(* Logix 5000 project; controller IF2_DEMO Emulate 5570 rev 20.12; software revision 20.04; part 4 of 8 *)
(* tags used below, declared in another part *)
   Alarm_Labeler1_Blocked : ALARM_DIGITAL;
   Alarm_Labeler1_Breakdown : ALARM_DIGITAL;
   Alarm_Labeler1_Starved : ALARM_DIGITAL;
   Alarm_Labeler1_Stopped : ALARM_DIGITAL;
   Blocked_Condition : BOOL;
   Breakdown_Labeler_Simulation : TIMER;
   Breakdown_Labeler_Simulator_Down_Switch : BOOL;
   Breakdown_Occurance_Time : DINT;
   Breakdown_Variation_Stepper : DINT;
   Expected_Full_Production_Rate : DINT;
   Labeler : FTVPDemoWorkCell;
   Labeler_Bottler_Per_Min : DINT;
   Labeler_Start : BOOL;
   Labeler_State : DINT;
   Labeler_Status : DINT;
   Labeler_Stop : BOOL;
   OEE_Availability : REAL;
   OEE_Overall : REAL;
   OEE_Performance : REAL;
   OEE_Quality : REAL;
   Starve_Block_Labeler_ONS : BOOL;
   Starved_Condition : BOOL;
   TempReadTrigger : TIMER;
   TempTimer : TIMER;
   TempTimer2 : TIMER;
   AlarmLabelJam : BOOL;
   ChangeOver_In_Progress : BOOL;
   Current_Order : STRING;
   CurrentCustomerName : STRING;
   CurrentPartName : STRING;
   DispenserLine : LineData;
   Filler_Bottles_Per_Minute : ALIAS FOR ProdCounts.Total;
   Filler_Stopped : BOOL;
   Labeler_Stopped : BOOL;
   OEE_Scrap_Labeler : DINT;
   OrderQty : DINT[4];
   Packaging_Stopped : BOOL;
   PartCountRollOver : DINT;
   Performance_Control : DINT;
   Previous_Order : STRING;
   PreviousCustomerName : STRING;
   PreviousPartName : STRING;
   ProdCounts : Counts;
   Product_Change : DINT;
   Production_Start_Labeler : BOOL;
   RefillLine : LineData;
   Starve_Block_Filler_Start_Toggle : BOOL;
   Starve_Block_Labeler_Start_Toggle : BOOL;
   Starve_Block_Packaging_Start_Toggle : BOOL;
   Timer1000ms : TIMER;
   Timer250ms : TIMER;
   WallClock : DINT[7];
   WC : WC[10];
(* LabelerD, continued *)

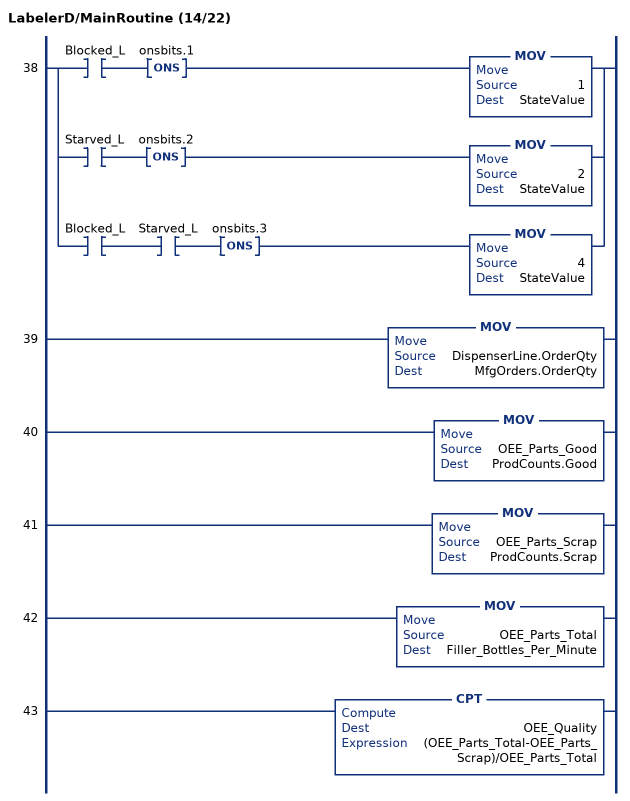
   38: [XIC(Blocked_L) ONS(onsbits.1) MOV(1,StateValue) ,XIC(Starved_L) ONS(onsbits.2) MOV(2,StateValue) ,XIC(Blocked_L) XIC(Starved_L) ONS(onsbits.3) MOV(4,StateValue) ];
   39: MOV(DispenserLine.OrderQty,MfgOrders.OrderQty);
   40: MOV(OEE_Parts_Good,ProdCounts.Good);
   41: MOV(OEE_Parts_Scrap,ProdCounts.Scrap);
   42: MOV(OEE_Parts_Total,Filler_Bottles_Per_Minute);
   43: CPT(OEE_Quality,(OEE_Parts_Total-OEE_Parts_Scrap)/OEE_Parts_Total);
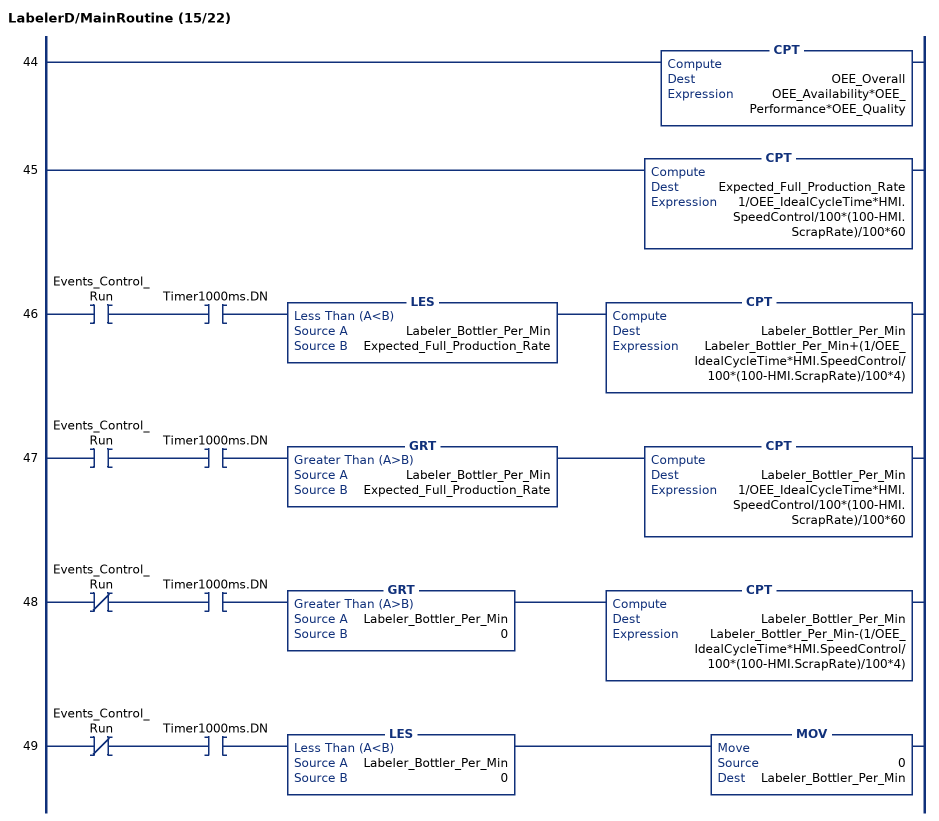
   44: CPT(OEE_Overall,OEE_Availability*OEE_Performance*OEE_Quality);
   45: CPT(Expected_Full_Production_Rate,1/OEE_IdealCycleTime*HMI.SpeedControl/100*(100-HMI.ScrapRate)/100*60);
   46: XIC(Events_Control_Run)XIC(Timer1000ms.DN)LES(Labeler_Bottler_Per_Min,Expected_Full_Production_Rate)CPT(Labeler_Bottler_Per_Min,Labeler_Bottler_Per_Min+(1/OEE_IdealCycleTime*HMI.SpeedControl/100*(100-HMI.ScrapRate)/100*4));
   47: XIC(Events_Control_Run)XIC(Timer1000ms.DN)GRT(Labeler_Bottler_Per_Min,Expected_Full_Production_Rate)CPT(Labeler_Bottler_Per_Min,1/OEE_IdealCycleTime*HMI.SpeedControl/100*(100-HMI.ScrapRate)/100*60);
   48: XIO(Events_Control_Run)XIC(Timer1000ms.DN)GRT(Labeler_Bottler_Per_Min,0)CPT(Labeler_Bottler_Per_Min,Labeler_Bottler_Per_Min-(1/OEE_IdealCycleTime*HMI.SpeedControl/100*(100-HMI.ScrapRate)/100*4));
   49: XIO(Events_Control_Run)XIC(Timer1000ms.DN)LES(Labeler_Bottler_Per_Min,0)MOV(0,Labeler_Bottler_Per_Min);
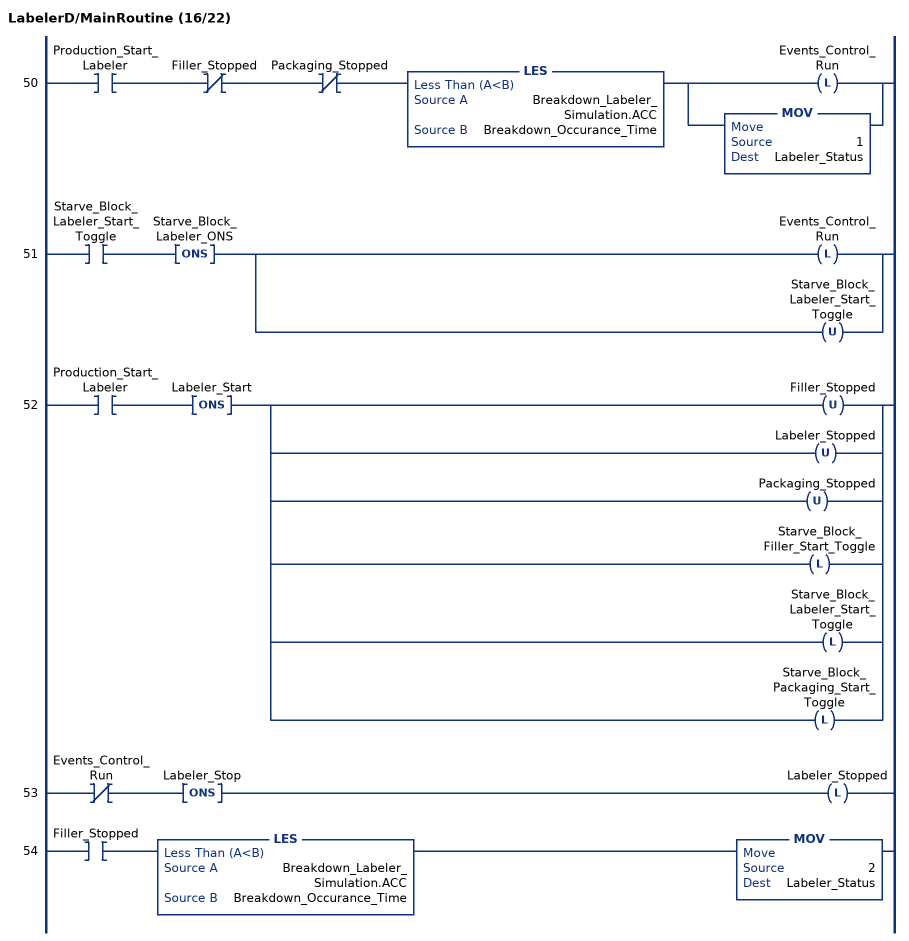
   50: XIC(Production_Start_Labeler)XIO(Filler_Stopped)XIO(Packaging_Stopped)LES(Breakdown_Labeler_Simulation.ACC,Breakdown_Occurance_Time)[OTL(Events_Control_Run) ,MOV(1,Labeler_Status) ];
   51: XIC(Starve_Block_Labeler_Start_Toggle)ONS(Starve_Block_Labeler_ONS)[OTL(Events_Control_Run) ,OTU(Starve_Block_Labeler_Start_Toggle) ];
   52: XIC(Production_Start_Labeler)ONS(Labeler_Start)[OTU(Filler_Stopped) ,OTU(Labeler_Stopped) ,OTU(Packaging_Stopped) ,OTL(Starve_Block_Filler_Start_Toggle) ,OTL(Starve_Block_Labeler_Start_Toggle) ,OTL(Starve_Block_Packaging_Start_Toggle) ];
   53: XIO(Events_Control_Run)ONS(Labeler_Stop)OTL(Labeler_Stopped);
   54: XIC(Filler_Stopped)LES(Breakdown_Labeler_Simulation.ACC,Breakdown_Occurance_Time)MOV(2,Labeler_Status);
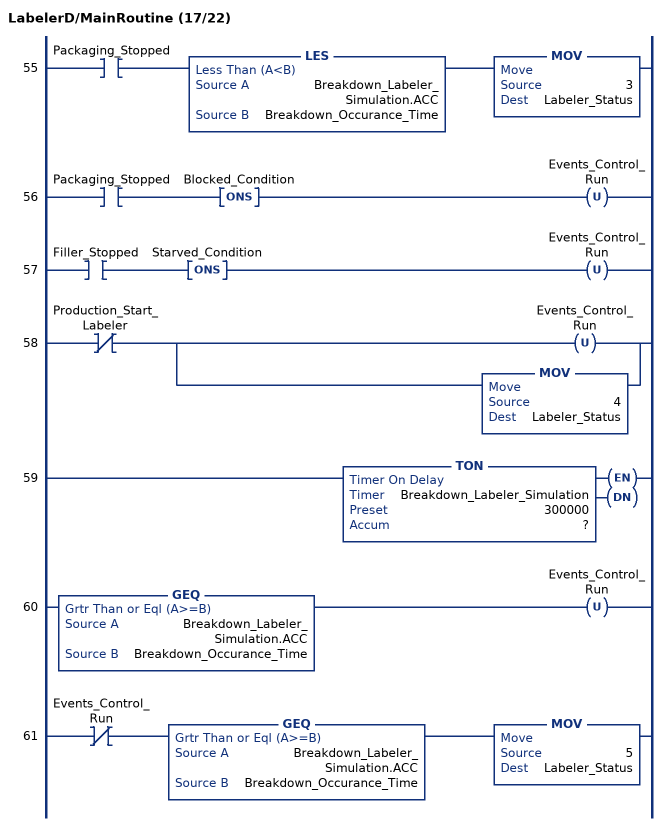
   55: XIC(Packaging_Stopped)LES(Breakdown_Labeler_Simulation.ACC,Breakdown_Occurance_Time)MOV(3,Labeler_Status);
   56: XIC(Packaging_Stopped)ONS(Blocked_Condition)OTU(Events_Control_Run);
   57: XIC(Filler_Stopped)ONS(Starved_Condition)OTU(Events_Control_Run);
   58: XIO(Production_Start_Labeler)[OTU(Events_Control_Run) ,MOV(4,Labeler_Status) ];
   59: TON(Breakdown_Labeler_Simulation,?,?);
   60: GEQ(Breakdown_Labeler_Simulation.ACC,Breakdown_Occurance_Time)OTU(Events_Control_Run);
   61: XIO(Events_Control_Run)GEQ(Breakdown_Labeler_Simulation.ACC,Breakdown_Occurance_Time)MOV(5,Labeler_Status);
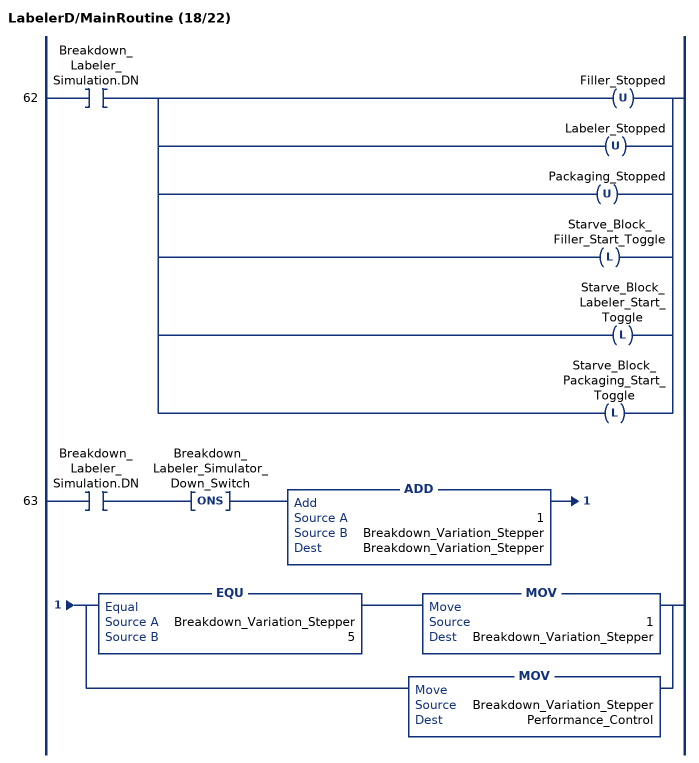
   62: XIC(Breakdown_Labeler_Simulation.DN)[OTU(Filler_Stopped) ,OTU(Labeler_Stopped) ,OTU(Packaging_Stopped) ,OTL(Starve_Block_Filler_Start_Toggle) ,OTL(Starve_Block_Labeler_Start_Toggle) ,OTL(Starve_Block_Packaging_Start_Toggle) ];
   63: XIC(Breakdown_Labeler_Simulation.DN)ONS(Breakdown_Labeler_Simulator_Down_Switch)ADD(1,Breakdown_Variation_Stepper,Breakdown_Variation_Stepper)[EQU(Breakdown_Variation_Stepper,5) MOV(1,Breakdown_Variation_Stepper) ,MOV(Breakdown_Variation_Stepper,Performance_Control) ];
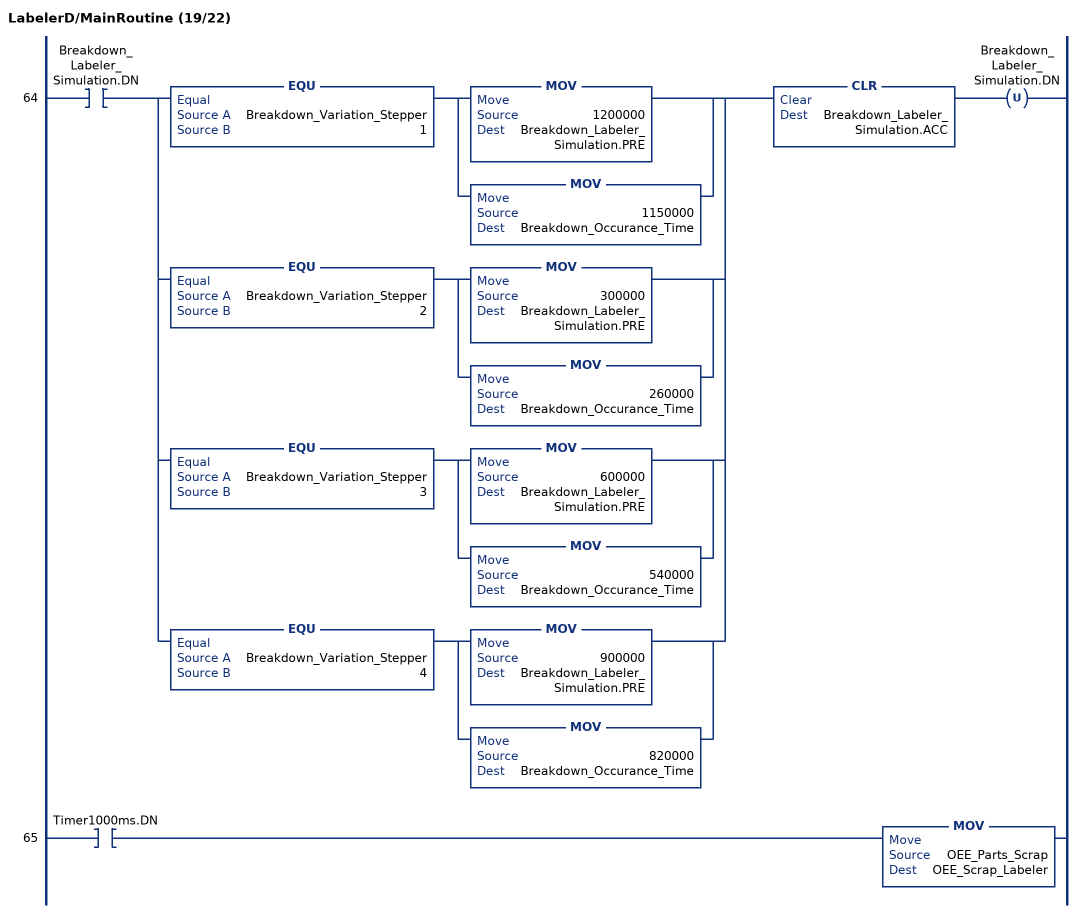
   64: XIC(Breakdown_Labeler_Simulation.DN)[EQU(Breakdown_Variation_Stepper,1) [MOV(1200000,Breakdown_Labeler_Simulation.PRE) ,MOV(1150000,Breakdown_Occurance_Time) ] ,EQU(Breakdown_Variation_Stepper,2) [MOV(300000,Breakdown_Labeler_Simulation.PRE) ,MOV(260000,Breakdown_Occurance_Time) ] ,EQU(Breakdown_Variation_Stepper,3) [MOV(600000,Breakdown_Labeler_Simulation.PRE) ,MOV(540000,Breakdown_Occurance_Time) ] ,EQU(Breakdown_Variation_Stepper,4) [MOV(900000,Breakdown_Labeler_Simulation.PRE) ,MOV(820000,Breakdown_Occurance_Time) ] ]CLR(Breakdown_Labeler_Simulation.ACC)OTU(Breakdown_Labeler_Simulation.DN);
   65: XIC(Timer1000ms.DN)MOV(OEE_Parts_Scrap,OEE_Scrap_Labeler);
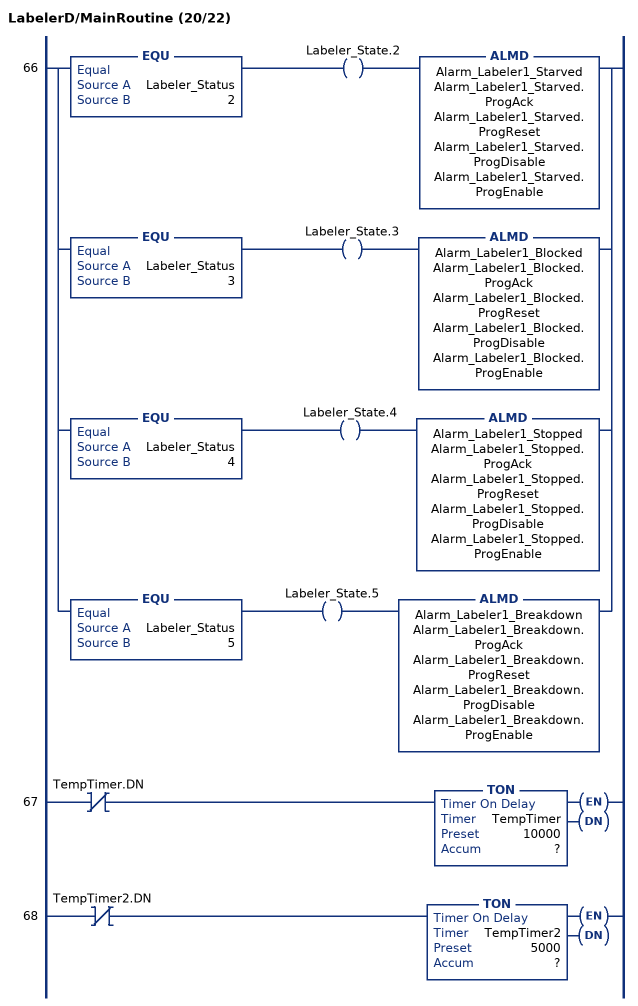
   66: [EQU(Labeler_Status,2) OTE(Labeler_State.2) ALMD(Alarm_Labeler1_Starved,Alarm_Labeler1_Starved.ProgAck,Alarm_Labeler1_Starved.ProgReset,Alarm_Labeler1_Starved.ProgDisable,Alarm_Labeler1_Starved.ProgEnable) ,EQU(Labeler_Status,3) OTE(Labeler_State.3) ALMD(Alarm_Labeler1_Blocked,Alarm_Labeler1_Blocked.ProgAck,Alarm_Labeler1_Blocked.ProgReset,Alarm_Labeler1_Blocked.ProgDisable,Alarm_Labeler1_Blocked.ProgEnable) ,EQU(Labeler_Status,4) OTE(Labeler_State.4) ALMD(Alarm_Labeler1_Stopped,Alarm_Labeler1_Stopped.ProgAck,Alarm_Labeler1_Stopped.ProgReset,Alarm_Labeler1_Stopped.ProgDisable,Alarm_Labeler1_Stopped.ProgEnable) ,EQU(Labeler_Status,5) OTE(Labeler_State.5) ALMD(Alarm_Labeler1_Breakdown,Alarm_Labeler1_Breakdown.ProgAck,Alarm_Labeler1_Breakdown.ProgReset,Alarm_Labeler1_Breakdown.ProgDisable,Alarm_Labeler1_Breakdown.ProgEnable) ];
   67: XIO(TempTimer.DN)TON(TempTimer,?,?);
   68: XIO(TempTimer2.DN)TON(TempTimer2,?,?);
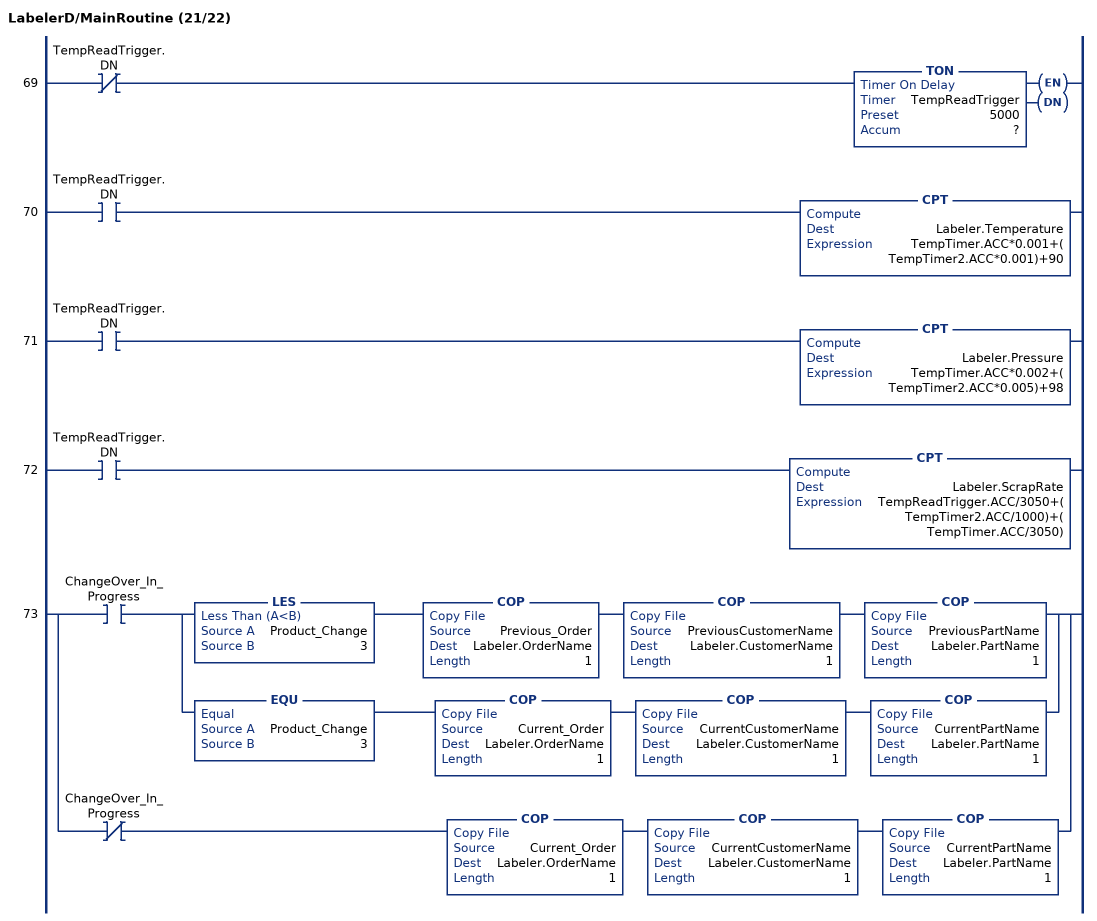
   69: XIO(TempReadTrigger.DN)TON(TempReadTrigger,?,?);
   70: XIC(TempReadTrigger.DN)CPT(Labeler.Temperature,TempTimer.ACC*0.001+(TempTimer2.ACC*0.001)+90);
   71: XIC(TempReadTrigger.DN)CPT(Labeler.Pressure,TempTimer.ACC*0.002+(TempTimer2.ACC*0.005)+98);
   72: XIC(TempReadTrigger.DN)CPT(Labeler.ScrapRate,TempReadTrigger.ACC/3050+(TempTimer2.ACC/1000)+(TempTimer.ACC/3050));
   73: [XIC(ChangeOver_In_Progress) [LES(Product_Change,3) COP(Previous_Order,Labeler.OrderName,1) COP(PreviousCustomerName,Labeler.CustomerName,1) COP(PreviousPartName,Labeler.PartName,1) ,EQU(Product_Change,3) COP(Current_Order,Labeler.OrderName,1) COP(CurrentCustomerName,Labeler.CustomerName,1) COP(CurrentPartName,Labeler.PartName,1) ] ,XIO(ChangeOver_In_Progress) COP(Current_Order,Labeler.OrderName,1) COP(CurrentCustomerName,Labeler.CustomerName,1) COP(CurrentPartName,Labeler.PartName,1) ];
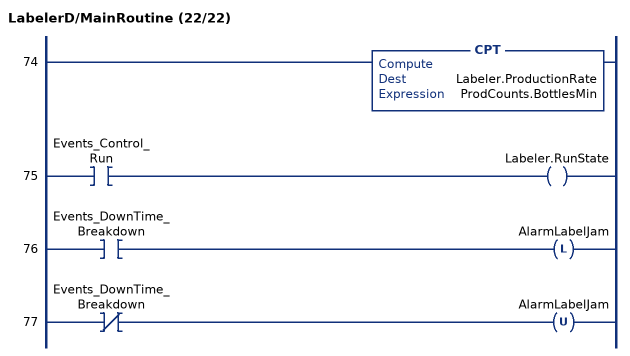
   74: CPT(Labeler.ProductionRate,ProdCounts.BottlesMin);
   75: XIC(Events_Control_Run)OTE(Labeler.RunState);
   76: XIC(Events_DownTime_Breakdown)OTL(AlarmLabelJam);
   77: XIO(Events_DownTime_Breakdown)OTU(AlarmLabelJam);
END_ROUTINE
END_PROGRAM

PROGRAM LabelerR   (* main routine MainRoutine *)
VAR
   Block_Delay : TIMER := (PRE := 15000);
   Blocked_L : BOOL;
   BottleCount : DINT := 298;
   BottleCounter : COUNTER := (PRE := 50000, ACC := 44);
   BottleMotion1 : TIMER := (PRE := 200, ACC := 15, EN := 1, TT := 1);
   Ctrl_Bit : BOOL := 1;
   Divisor1 : DINT := 5;
   DownStream_Run : ALIAS FOR WC[9].EventTrigger[0].1;
   DownStream_Running : ALIAS FOR WC[9].EventTrigger[0].8;
   Events : Events := (DownTime.BreakdownCode := 5, Control.StandbyCode := 1, Control.Run := 1, Control.Auto := 1);
   Events_Control_Auto : ALIAS FOR WC_L.EventTrigger[0].5;
   Events_Control_OpStop : ALIAS FOR WC_L.EventTrigger[0].3;
   Events_Control_Run : ALIAS FOR WC_L.EventTrigger[0].1;
   Events_Control_Running : ALIAS FOR WC_L.EventTrigger[0].8;
   Events_Control_Standby : ALIAS FOR WC_L.EventTrigger[0].0;
   Events_Control_StandbyCode : ALIAS FOR WC_L.EventValue_REAL[1];
   Events_DownTime_Breakdown : ALIAS FOR WC_L.EventTrigger[0].2;
   Events_DownTime_BreakdownCode : ALIAS FOR WC_L.EventValue_REAL[2];
   Events_DownTime_Testing : ALIAS FOR WC_L.EventTrigger[0].7;
   Events_DownTime_UnschedMaint : ALIAS FOR WC_L.EventTrigger[0].6;
   Events_Operate_Load : ALIAS FOR WC_L.EventTrigger[0].10;
   Events_Operate_OrderProc : ALIAS FOR WC_L.EventTrigger[0].11;
   Events_Operate_Setup : ALIAS FOR WC_L.EventTrigger[0].9;
   HMI : HMIVars := (ScrapRate := 5.0, SpeedControl := 100.0, PrevSpeed := 100.0, PartCountRollOver := 9999999, MfgTimeBase := 1, MaxEventDur := 12.0, MinEventDur := 7.0, EventsPerHr := 55, EventDur := 11.992554, RunDur := 52.29316, MinRunDur := 5.0);
   MfgOrders : MfgOrders := (CustomerName := 'Big-Mart', OrderName := 'C321', OrderQty := 30000, ProdRate := 60.0, SetupTime := 8.0, PartName := 'STRAW-R40', WorkcellName := 'LabelerR', PartNameSav := 'STRAW-R40');
   MfgOrders_CustomerName : ALIAS FOR WC_L.FlexSTRING[4];
   MfgOrders_OrderName : ALIAS FOR WC_L.FlexSTRING[3];
   MfgOrders_PartName : ALIAS FOR WC_L.FlexSTRING[0];
   Motion : DINT := 70;
   Motion1Bit : BOOL := 1;
   Motion_Counter : DINT := 1;
   Motion_Speed : DINT := 10;
   MotionCount : TIMER := (PRE := 900);
   MotionHolder1 : DINT := 37;
   OEE : OEE := (IdealCycleTime := 4.0);
   OEE_IdealCycleTime : ALIAS FOR WC_L.IdealCT;
   OEE_Parts_Good : ALIAS FOR WC_L.GoodParts;
   OEE_Parts_Scrap : ALIAS FOR WC_L.ScrapParts;
   OEE_Parts_Total : ALIAS FOR WC_L.TotalParts;
   onsbits : DINT;
   OperatorID : ALIAS FOR WC_L.FlexREAL[1];
   Pressure1 : ALIAS FOR WC_L.PV[0];   // PSI
   ProductColorCode : INT := 3;
   Reset1Bit : BOOL;
   SecondTimer : TIMER := (PRE := 60000, ACC := 8946, EN := 1, TT := 1);
   SIM : SimVars := (Run.PRE := 52293, Event.PRE := 7000, Setup.PRE := 7000, EventNumber := 2, UtilityBool[2] := 1);
        .UTILITYBOOL[2]   // First Scan Bit
   Starve_Delay : TIMER := (PRE := 15000);
   Starved_L : BOOL;
   StateValue : ALIAS FOR WC_L.MonitorValue[0];
   Suppress : Events;
   Temperature1 : ALIAS FOR WC_L.PV[1];   // DEG
   UpStream_Run : ALIAS FOR WC[3].EventTrigger[0].1;
   UpStream_Running : ALIAS FOR WC[3].EventTrigger[0].8;
   WC_L : ALIAS FOR WC[5];
END_VAR

ROUTINE MainRoutine   (* ladder *)
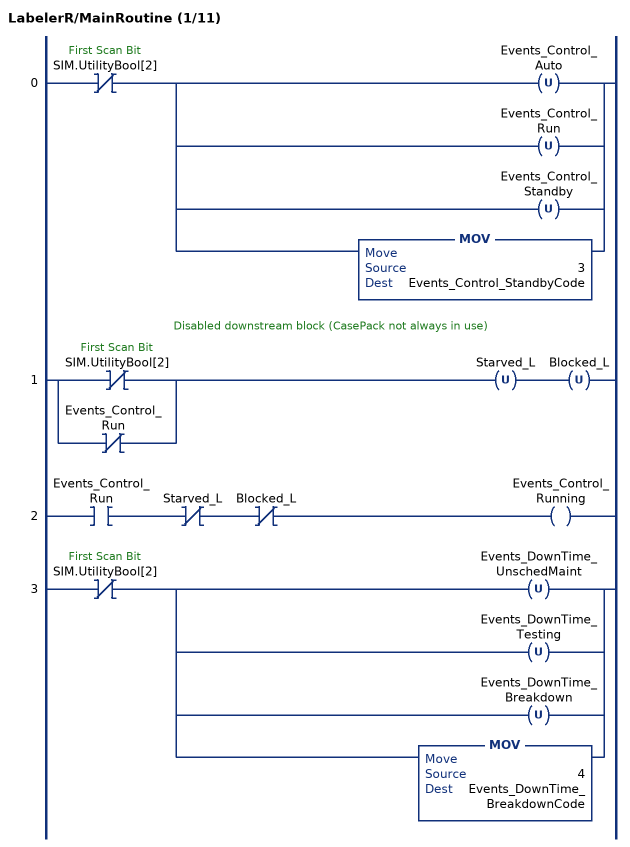
   0: XIO(SIM.UtilityBool[2])[OTU(Events_Control_Auto) ,OTU(Events_Control_Run) ,OTU(Events_Control_Standby) ,MOV(3,Events_Control_StandbyCode) ];
   // Disabled downstream block (CasePack not always in use)
   1: [XIO(SIM.UtilityBool[2]) ,XIO(Events_Control_Run) ]OTU(Starved_L)OTU(Blocked_L);
   2: XIC(Events_Control_Run)XIO(Starved_L)XIO(Blocked_L)OTE(Events_Control_Running);
   3: XIO(SIM.UtilityBool[2])[OTU(Events_DownTime_UnschedMaint) ,OTU(Events_DownTime_Testing) ,OTU(Events_DownTime_Breakdown) ,MOV(4,Events_DownTime_BreakdownCode) ];
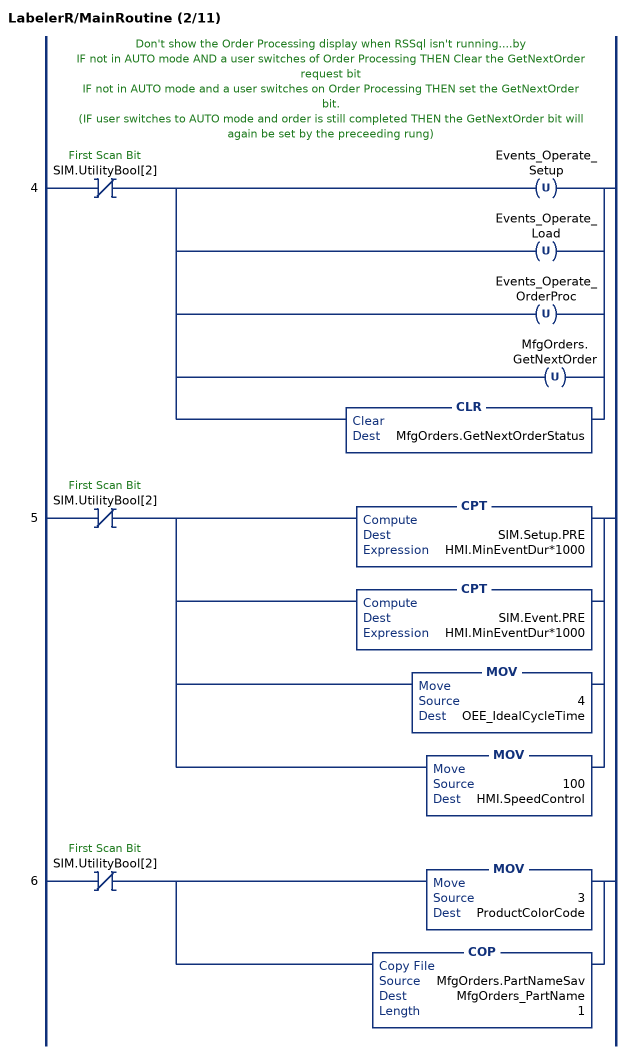
   // Don't show the Order Processing display when RSSql isn't running....by
   // IF not in AUTO mode AND a user switches of Order Processing THEN Clear the GetNextOrder request bit
   // IF not in AUTO mode and a user switches on Order Processing THEN set the GetNextOrder bit.
   // (IF user switches to AUTO mode and order is still completed THEN the GetNextOrder bit will again be set by the preceeding rung)
   4: XIO(SIM.UtilityBool[2])[OTU(Events_Operate_Setup) ,OTU(Events_Operate_Load) ,OTU(Events_Operate_OrderProc) ,OTU(MfgOrders.GetNextOrder) ,CLR(MfgOrders.GetNextOrderStatus) ];
   5: XIO(SIM.UtilityBool[2])[CPT(SIM.Setup.PRE,HMI.MinEventDur*1000) ,CPT(SIM.Event.PRE,HMI.MinEventDur*1000) ,MOV(4,OEE_IdealCycleTime) ,MOV(100,HMI.SpeedControl) ];
   6: XIO(SIM.UtilityBool[2])[MOV(3,ProductColorCode) ,COP(MfgOrders.PartNameSav,MfgOrders_PartName,1) ];
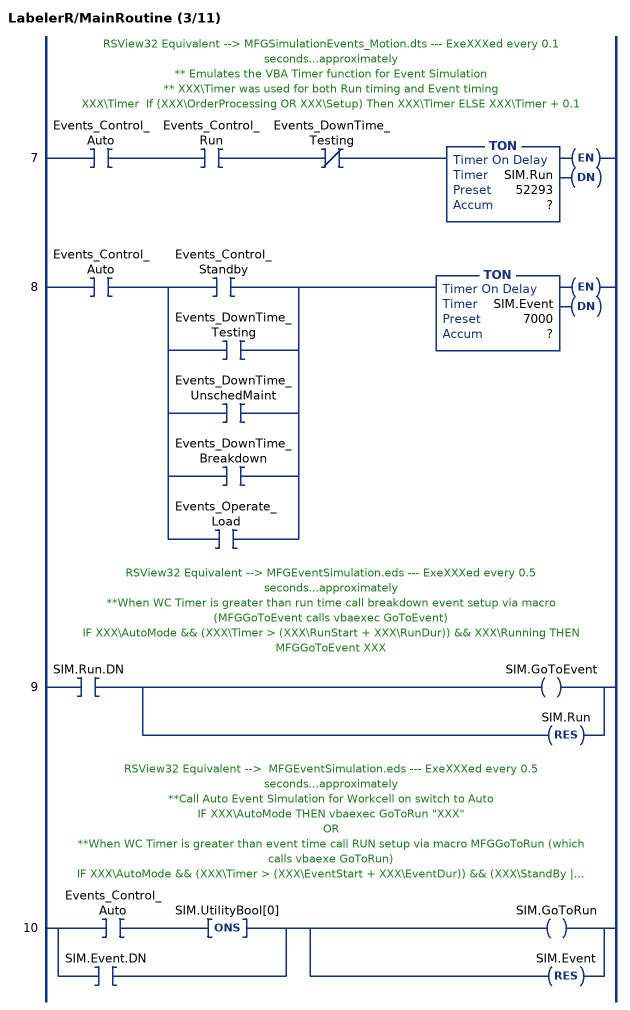
   // RSView32 Equivalent --> MFGSimulationEvents_Motion.dts --- ExeXXXed every 0.1 seconds...approximately
   // ** Emulates the VBA Timer function for Event Simulation
   // ** XXX\Timer was used for both Run timing and Event timing
   // XXX\Timer	If (XXX\OrderProcessing OR XXX\Setup) Then XXX\Timer ELSE XXX\Timer + 0.1
   7: XIC(Events_Control_Auto)XIC(Events_Control_Run)XIO(Events_DownTime_Testing)TON(SIM.Run,?,?);
   8: XIC(Events_Control_Auto)[XIC(Events_Control_Standby) ,XIC(Events_DownTime_Testing) ,XIC(Events_DownTime_UnschedMaint) ,XIC(Events_DownTime_Breakdown) ,XIC(Events_Operate_Load) ]TON(SIM.Event,?,?);
   // RSView32 Equivalent --> MFGEventSimulation.eds --- ExeXXXed every 0.5 seconds...approximately
   // **When WC Timer is greater than run time call breakdown event setup via macro (MFGGoToEvent calls vbaexec GoToEvent)
   // IF XXX\AutoMode && (XXX\Timer > (XXX\RunStart + XXX\RunDur)) && XXX\Running THEN MFGGoToEvent XXX
   9: XIC(SIM.Run.DN)[OTE(SIM.GoToEvent) ,RES(SIM.Run) ];
   // RSView32 Equivalent -->  MFGEventSimulation.eds --- ExeXXXed every 0.5 seconds...approximately
   // **Call Auto Event Simulation for Workcell on switch to Auto
   // IF XXX\AutoMode THEN vbaexec GoToRun "XXX"
   // OR
   // **When WC Timer is greater than event time call RUN setup via macro MFGGoToRun (which calls vbaexe GoToRun)
   // IF XXX\AutoMode && (XXX\Timer > (XXX\EventStart + XXX\EventDur)) && (XXX\StandBy || XXX\Test || XXX\UnSchedMaint || XXX\Breakdown ||XXX\Load) THEN MFGGoToRun XXX
   10: [XIC(Events_Control_Auto) ONS(SIM.UtilityBool[0]) ,XIC(SIM.Event.DN) ][OTE(SIM.GoToRun) ,RES(SIM.Event) ];
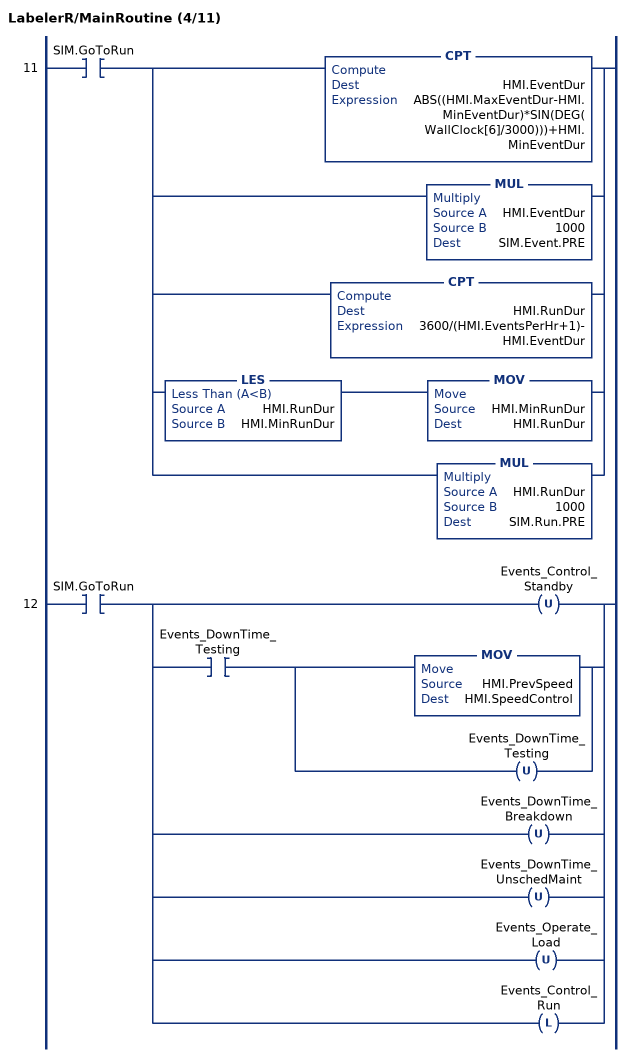
   11: XIC(SIM.GoToRun)[CPT(HMI.EventDur,ABS((HMI.MaxEventDur-HMI.MinEventDur)*SIN(DEG(WallClock[6]/3000)))+HMI.MinEventDur) ,MUL(HMI.EventDur,1000,SIM.Event.PRE) ,CPT(HMI.RunDur,3600/(HMI.EventsPerHr+1)-HMI.EventDur) ,LES(HMI.RunDur,HMI.MinRunDur) MOV(HMI.MinRunDur,HMI.RunDur) ,MUL(HMI.RunDur,1000,SIM.Run.PRE) ];
   12: XIC(SIM.GoToRun)[OTU(Events_Control_Standby) ,XIC(Events_DownTime_Testing) [MOV(HMI.PrevSpeed,HMI.SpeedControl) ,OTU(Events_DownTime_Testing) ] ,OTU(Events_DownTime_Breakdown) ,OTU(Events_DownTime_UnschedMaint) ,OTU(Events_Operate_Load) ,OTL(Events_Control_Run) ];
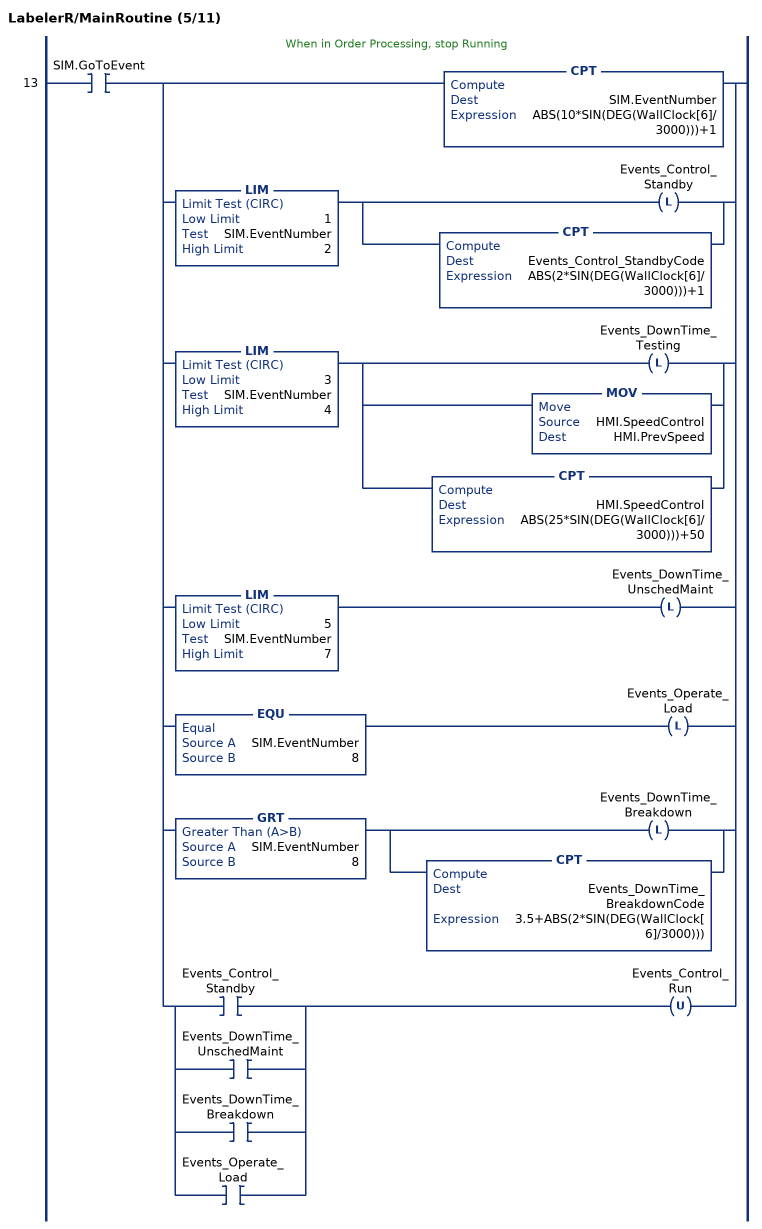
   // When in Order Processing, stop Running
   13: XIC(SIM.GoToEvent)[CPT(SIM.EventNumber,ABS(10*SIN(DEG(WallClock[6]/3000)))+1) ,LIM(1,SIM.EventNumber,2) [OTL(Events_Control_Standby) ,CPT(Events_Control_StandbyCode,ABS(2*SIN(DEG(WallClock[6]/3000)))+1) ] ,LIM(3,SIM.EventNumber,4) [OTL(Events_DownTime_Testing) ,MOV(HMI.SpeedControl,HMI.PrevSpeed) ,CPT(HMI.SpeedControl,ABS(25*SIN(DEG(WallClock[6]/3000)))+50) ] ,LIM(5,SIM.EventNumber,7) OTL(Events_DownTime_UnschedMaint) ,EQU(SIM.EventNumber,8) OTL(Events_Operate_Load) ,GRT(SIM.EventNumber,8) [OTL(Events_DownTime_Breakdown) ,CPT(Events_DownTime_BreakdownCode,3.5+ABS(2*SIN(DEG(WallClock[6]/3000)))) ] ,[XIC(Events_Control_Standby) ,XIC(Events_DownTime_UnschedMaint) ,XIC(Events_DownTime_Breakdown) ,XIC(Events_Operate_Load) ] OTU(Events_Control_Run) ];
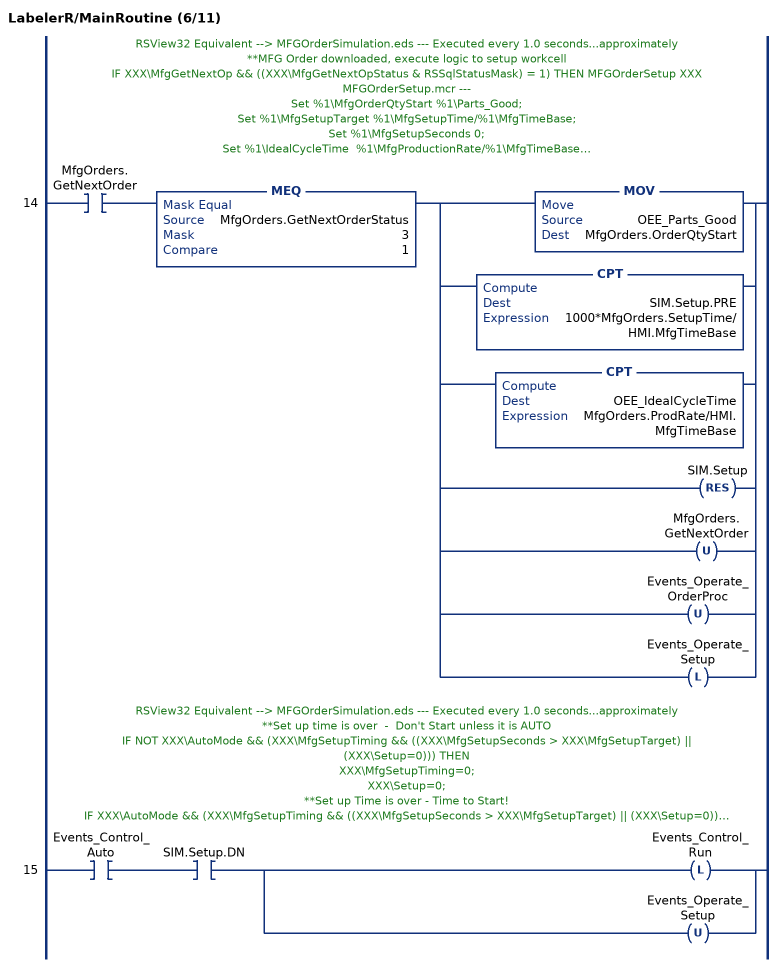
   // RSView32 Equivalent --> MFGOrderSimulation.eds --- Executed every 1.0 seconds...approximately
   // **MFG Order downloaded, execute logic to setup workcell
   // IF XXX\MfgGetNextOp && ((XXX\MfgGetNextOpStatus & RSSqlStatusMask) = 1) THEN MFGOrderSetup XXX
   // MFGOrderSetup.mcr ---
   // 	Set %1\MfgOrderQtyStart %1\Parts_Good;
   // 	Set %1\MfgSetupTarget %1\MfgSetupTime/%1\MfgTimeBase;
   // 	Set %1\MfgSetupSeconds 0;
   // 	Set %1\IdealCycleTime  %1\MfgProductionRate/%1\MfgTimeBase;
   // 	Set %1\MfgGetNextOp 0;
   // 	Set %1\Setup 1;
   // 	Set %1\OrderProcessing 0;
   // 	Set %1\MfgSetupTiming 1;
   14: XIC(MfgOrders.GetNextOrder)MEQ(MfgOrders.GetNextOrderStatus,3,1)[MOV(OEE_Parts_Good,MfgOrders.OrderQtyStart) ,CPT(SIM.Setup.PRE,1000*MfgOrders.SetupTime/HMI.MfgTimeBase) ,CPT(OEE_IdealCycleTime,MfgOrders.ProdRate/HMI.MfgTimeBase) ,RES(SIM.Setup) ,OTU(MfgOrders.GetNextOrder) ,OTU(Events_Operate_OrderProc) ,OTL(Events_Operate_Setup) ];
   // RSView32 Equivalent --> MFGOrderSimulation.eds --- Executed every 1.0 seconds...approximately
   // **Set up time is over  -  Don't Start unless it is AUTO
   // IF NOT XXX\AutoMode && (XXX\MfgSetupTiming && ((XXX\MfgSetupSeconds > XXX\MfgSetupTarget) || (XXX\Setup=0))) THEN
   // 	XXX\MfgSetupTiming=0;
   // 	XXX\Setup=0;
   // **Set up Time is over - Time to Start!
   // IF XXX\AutoMode && (XXX\MfgSetupTiming && ((XXX\MfgSetupSeconds > XXX\MfgSetupTarget) || (XXX\Setup=0))) THEN
   // 	XXX\MfgSetupTiming=0;
   // 	XXX\Setup=0;
   // 	XXX\RUNNING=1
   15: XIC(Events_Control_Auto)XIC(SIM.Setup.DN)[OTL(Events_Control_Run) ,OTU(Events_Operate_Setup) ];
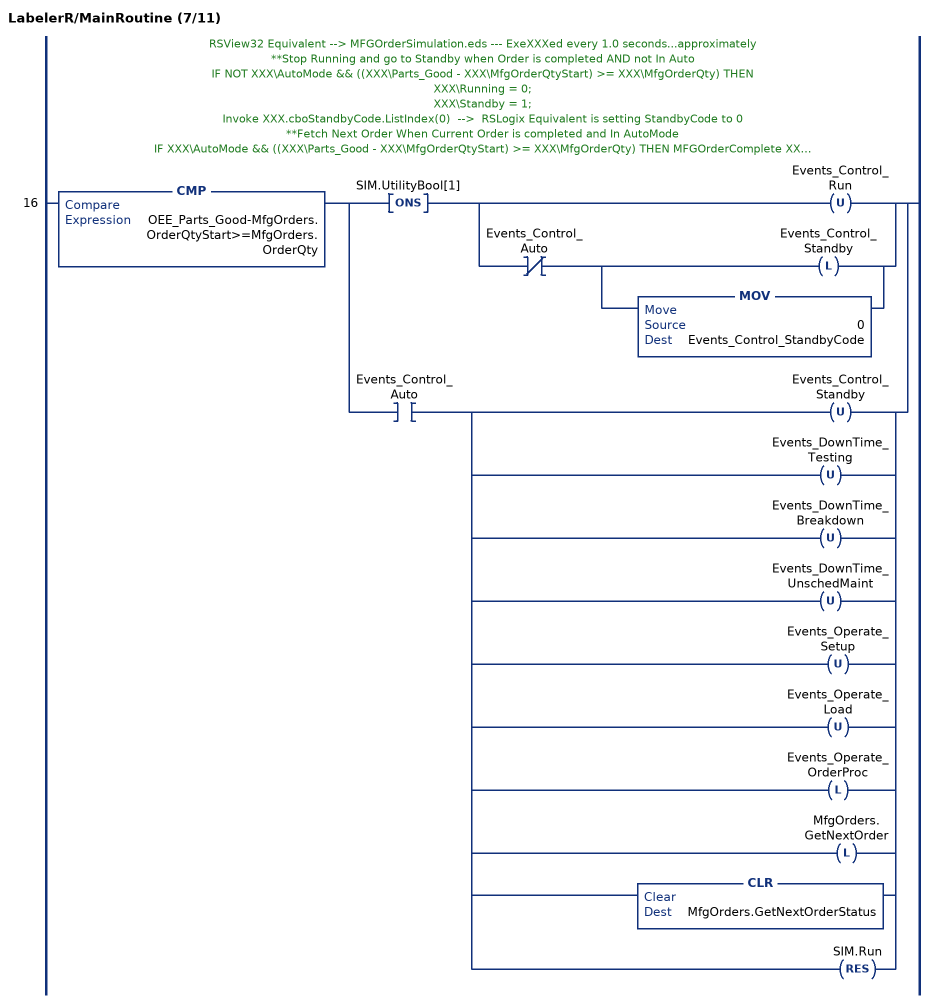
   // RSView32 Equivalent --> MFGOrderSimulation.eds --- ExeXXXed every 1.0 seconds...approximately
   // **Stop Running and go to Standby when Order is completed AND not In Auto
   // IF NOT XXX\AutoMode && ((XXX\Parts_Good - XXX\MfgOrderQtyStart) >= XXX\MfgOrderQty) THEN
   // 	XXX\Running = 0;
   // 	XXX\Standby = 1;
   // 	Invoke XXX.cboStandbyCode.ListIndex(0)  -->  RSLogix Equivalent is setting StandbyCode to 0
   // **Fetch Next Order When Current Order is completed and In AutoMode
   // IF XXX\AutoMode && ((XXX\Parts_Good - XXX\MfgOrderQtyStart) >= XXX\MfgOrderQty) THEN MFGOrderComplete XXX
   // MFGOrderComplete.mcr --- (Macros exeXXXed when called. %1 is the Workcell name -- typical all mcrs)
   // 	Set %1\RunStart %1\Timer;
   // 	Set %1\StandBy 0;
   // 	Set %1\Test 0;
   // 	Set %1\UnSchedMaint 0;
   // 	Set %1\Breakdown 0;
   // 	Set %1\Load 0;
   // 	Set %1\OrderProcessing 1;
   // 	Set %1\Running 0;
   // 	Set %1\MFGGetNextOpStatus 0;
   // 	Set %1\MFGGetNextOp 1
   16: CMP(OEE_Parts_Good-MfgOrders.OrderQtyStart>=MfgOrders.OrderQty)[ONS(SIM.UtilityBool[1]) [OTU(Events_Control_Run) ,XIO(Events_Control_Auto) [OTL(Events_Control_Standby) ,MOV(0,Events_Control_StandbyCode) ] ] ,XIC(Events_Control_Auto) [OTU(Events_Control_Standby) ,OTU(Events_DownTime_Testing) ,OTU(Events_DownTime_Breakdown) ,OTU(Events_DownTime_UnschedMaint) ,OTU(Events_Operate_Setup) ,OTU(Events_Operate_Load) ,OTL(Events_Operate_OrderProc) ,OTL(MfgOrders.GetNextOrder) ,CLR(MfgOrders.GetNextOrderStatus) ,RES(SIM.Run) ] ];
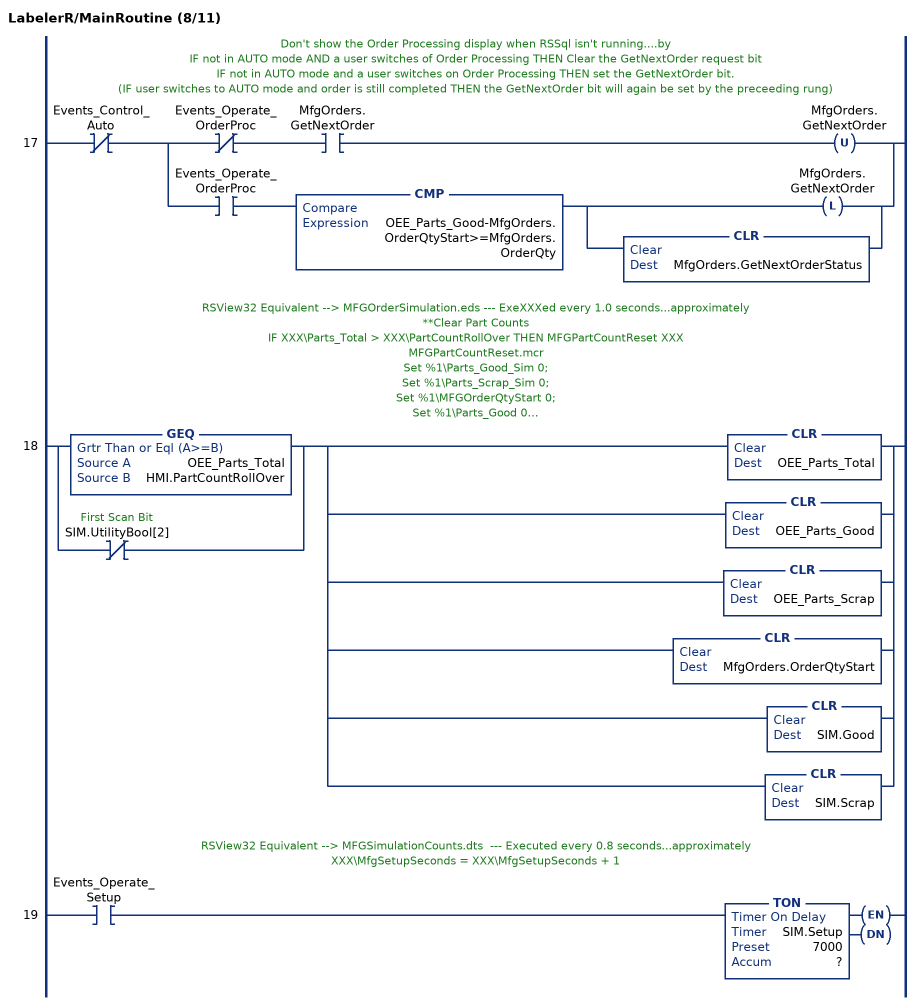
   // Don't show the Order Processing display when RSSql isn't running....by
   // IF not in AUTO mode AND a user switches of Order Processing THEN Clear the GetNextOrder request bit
   // IF not in AUTO mode and a user switches on Order Processing THEN set the GetNextOrder bit.
   // (IF user switches to AUTO mode and order is still completed THEN the GetNextOrder bit will again be set by the preceeding rung)
   17: XIO(Events_Control_Auto)[XIO(Events_Operate_OrderProc) XIC(MfgOrders.GetNextOrder) OTU(MfgOrders.GetNextOrder) ,XIC(Events_Operate_OrderProc) CMP(OEE_Parts_Good-MfgOrders.OrderQtyStart>=MfgOrders.OrderQty) [OTL(MfgOrders.GetNextOrder) ,CLR(MfgOrders.GetNextOrderStatus) ] ];
   // RSView32 Equivalent --> MFGOrderSimulation.eds --- ExeXXXed every 1.0 seconds...approximately
   // **Clear Part Counts
   // IF XXX\Parts_Total > XXX\PartCountRollOver THEN MFGPartCountReset XXX
   // MFGPartCountReset.mcr
   // 	Set %1\Parts_Good_Sim 0;
   // 	Set %1\Parts_Scrap_Sim 0;
   // 	Set %1\MFGOrderQtyStart 0;
   // 	Set %1\Parts_Good 0;
   // 	Set %1\Parts_Scrap 0;
   // 	Set %1\Parts_Total 0
   18: [GEQ(OEE_Parts_Total,HMI.PartCountRollOver) ,XIO(SIM.UtilityBool[2]) ][CLR(OEE_Parts_Total) ,CLR(OEE_Parts_Good) ,CLR(OEE_Parts_Scrap) ,CLR(MfgOrders.OrderQtyStart) ,CLR(SIM.Good) ,CLR(SIM.Scrap) ];
   // RSView32 Equivalent --> MFGSimulationCounts.dts	--- Executed every 0.8 seconds...approximately
   // XXX\MfgSetupSeconds = XXX\MfgSetupSeconds + 1
   19: XIC(Events_Operate_Setup)TON(SIM.Setup,?,?);
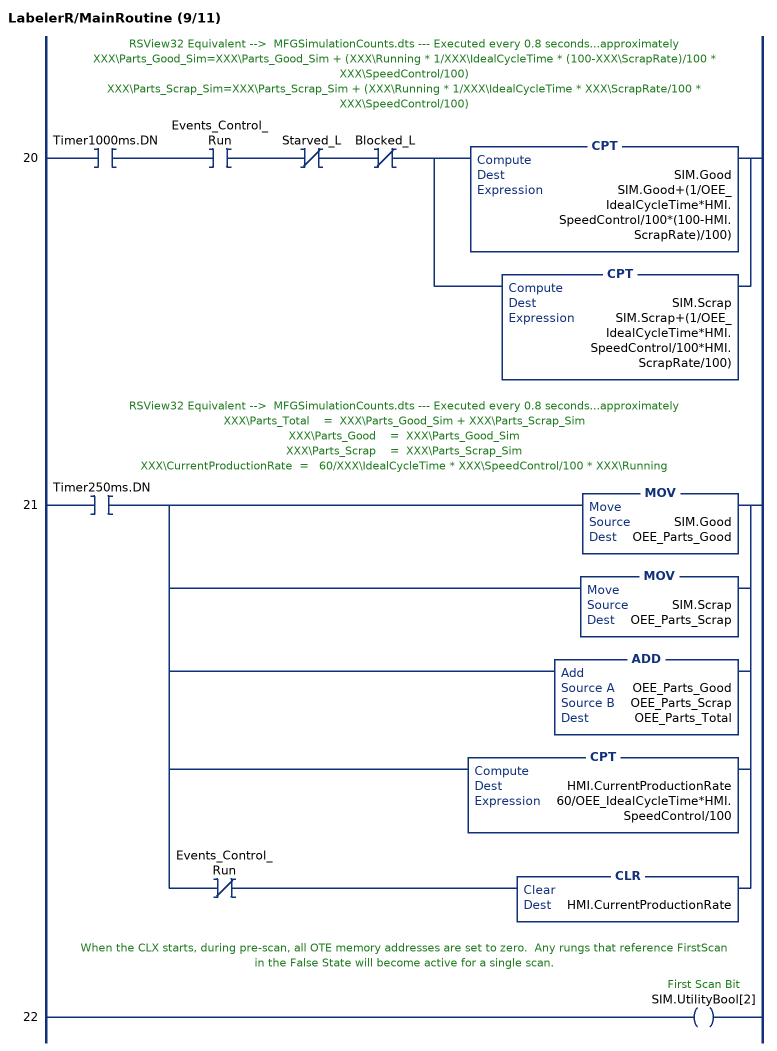
   // RSView32 Equivalent -->  MFGSimulationCounts.dts --- Executed every 0.8 seconds...approximately
   // XXX\Parts_Good_Sim=XXX\Parts_Good_Sim + (XXX\Running * 1/XXX\IdealCycleTime * (100-XXX\ScrapRate)/100 * XXX\SpeedControl/100)
   // XXX\Parts_Scrap_Sim=XXX\Parts_Scrap_Sim + (XXX\Running * 1/XXX\IdealCycleTime * XXX\ScrapRate/100 * XXX\SpeedControl/100)
   20: XIC(Timer1000ms.DN)XIC(Events_Control_Run)XIO(Starved_L)XIO(Blocked_L)[CPT(SIM.Good,SIM.Good+(1/OEE_IdealCycleTime*HMI.SpeedControl/100*(100-HMI.ScrapRate)/100)) ,CPT(SIM.Scrap,SIM.Scrap+(1/OEE_IdealCycleTime*HMI.SpeedControl/100*HMI.ScrapRate/100)) ];
   // RSView32 Equivalent -->  MFGSimulationCounts.dts --- Executed every 0.8 seconds...approximately
   // XXX\Parts_Total		=	XXX\Parts_Good_Sim + XXX\Parts_Scrap_Sim
   // XXX\Parts_Good		=	XXX\Parts_Good_Sim
   // XXX\Parts_Scrap		=	XXX\Parts_Scrap_Sim
   // XXX\CurrentProductionRate  = 	60/XXX\IdealCycleTime * XXX\SpeedControl/100 * XXX\Running
   21: XIC(Timer250ms.DN)[[MOV(SIM.Good,OEE_Parts_Good) ,MOV(SIM.Scrap,OEE_Parts_Scrap) ,ADD(OEE_Parts_Good,OEE_Parts_Scrap,OEE_Parts_Total) ] ,CPT(HMI.CurrentProductionRate,60/OEE_IdealCycleTime*HMI.SpeedControl/100) ,XIO(Events_Control_Run) CLR(HMI.CurrentProductionRate) ];
   // When the CLX starts, during pre-scan, all OTE memory addresses are set to zero.  Any rungs that reference FirstScan in the False State will become active for a single scan.
   22: OTE(SIM.UtilityBool[2]);
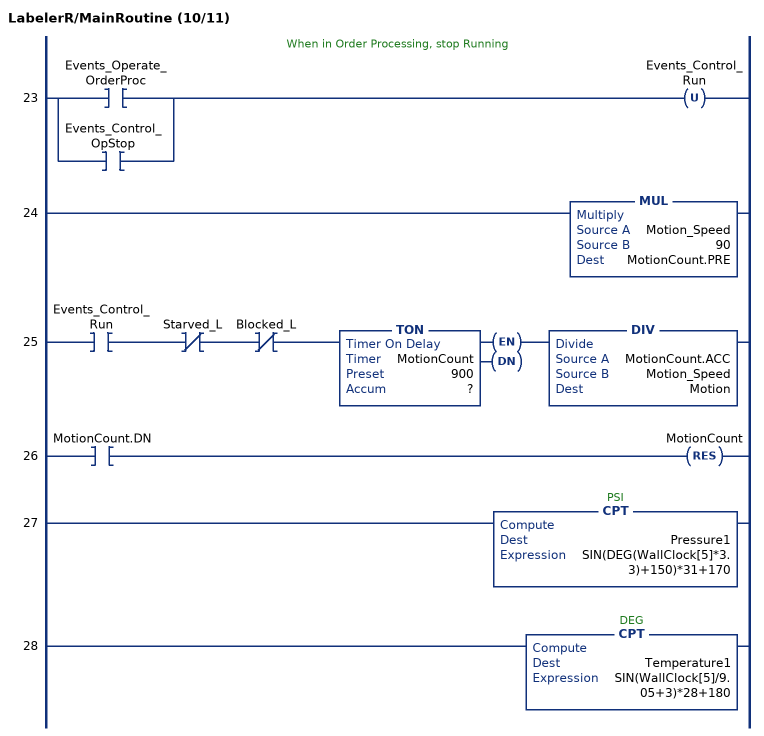
   // When in Order Processing, stop Running
   23: [XIC(Events_Operate_OrderProc) ,XIC(Events_Control_OpStop) ]OTU(Events_Control_Run);
   24: MUL(Motion_Speed,90,MotionCount.PRE);
   25: XIC(Events_Control_Run)XIO(Starved_L)XIO(Blocked_L)TON(MotionCount,?,?)DIV(MotionCount.ACC,Motion_Speed,Motion);
   26: XIC(MotionCount.DN)RES(MotionCount);
   27: CPT(Pressure1,SIN(DEG(WallClock[5]*3.3)+150)*31+170);
   28: CPT(Temperature1,SIN(WallClock[5]/9.05+3)*28+180);
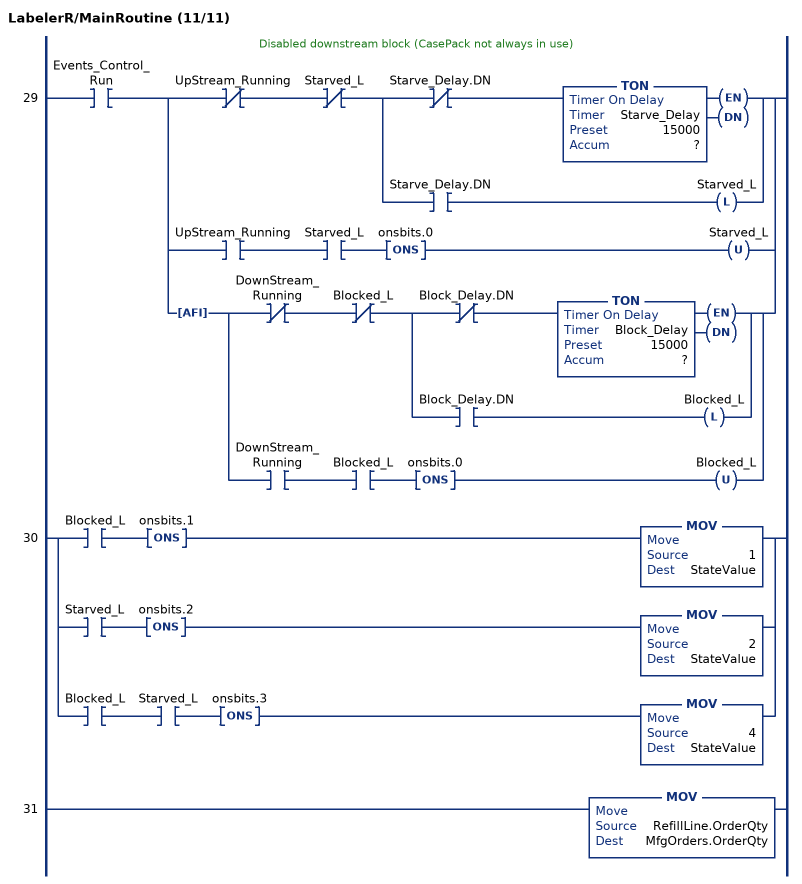
   // Disabled downstream block (CasePack not always in use)
   29: XIC(Events_Control_Run)[[XIO(UpStream_Running) XIO(Starved_L) [XIO(Starve_Delay.DN) TON(Starve_Delay,?,?) ,XIC(Starve_Delay.DN) OTL(Starved_L) ] ,XIC(UpStream_Running) XIC(Starved_L) ONS(onsbits.0) OTU(Starved_L) ] ,AFI() [XIO(DownStream_Running) XIO(Blocked_L) [XIO(Block_Delay.DN) TON(Block_Delay,?,?) ,XIC(Block_Delay.DN) OTL(Blocked_L) ] ,XIC(DownStream_Running) XIC(Blocked_L) ONS(onsbits.0) OTU(Blocked_L) ] ];
   30: [XIC(Blocked_L) ONS(onsbits.1) MOV(1,StateValue) ,XIC(Starved_L) ONS(onsbits.2) MOV(2,StateValue) ,XIC(Blocked_L) XIC(Starved_L) ONS(onsbits.3) MOV(4,StateValue) ];
   31: MOV(RefillLine.OrderQty,MfgOrders.OrderQty);
END_ROUTINE
END_PROGRAM
